PROGRAM MAIN
VAR
END_VAR

END_PROGRAM

(* stored: Version 1.1.0.1
   POU MAIN: Id {73c71207-fd27-47f6-8a77-50fd2fbb8782} *)
